INTERFACE IPistonGripper

METHOD Close : TcoCore.ITcoTaskStatus
END_METHOD

METHOD Open : TcoCore.ITcoTaskStatus
END_METHOD

END_INTERFACE

(* stored: Version 1.1.0.1, ProductVersion 3.1.4024.9
   Itf IPistonGripper: Id {53ede753-5654-0d31-350c-a0193aaffe9b}
   Folder Gripper: Id {4afb1eef-5dbf-0534-0f1e-a33213766255}
   Method Close: Id {f8b7dab3-47d6-090c-1f62-55767e5cccdf}
   Method Open: Id {6be1af67-892e-0d4d-260e-4e26f06d4807} *)
